VISUALIZATION PageAuto  // 1500x860
END_VISUALIZATION

(* stored: Version 1.1.0.1, ProductVersion 3.1.4024.9
   Visu PageAuto: Id {a8b44197-37b9-486e-87d8-5bb5cbfcd2d4} *)
